{attribute 'qualified_only'}
VAR_GLOBAL
END_VAR

(* stored: Version 1.1.0.1, ProductVersion 3.1.4024.9
   GVL GVL_2: Id {b8afa809-405b-4f4b-b509-33d76288af52} *)
